(* PLC project  *)

PROGRAM P

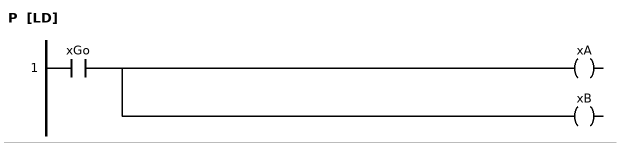
(* LD diagram, written out as Structured Text *)
xA := xGo;
xB := xGo;
END_PROGRAM
